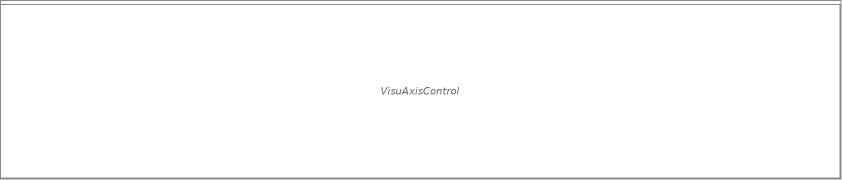
VISUALIZATION VisuAxisX  // 842x180
    Frame (0,4 840x174)
        shows VisuAxisControl(sAxisName := sAxisXName, stAxisVisu := stAxisX)
END_VISUALIZATION

(* stored: Version 1.1.0.1, ProductVersion 3.1.4022.6
   Visu VisuAxisX: Id {03ecdd57-fc88-48f1-a1c2-cde9123672ff} *)
